HMI tags "Default tag table"
   "DB500_SinaisIhm_ManFrente" : Bool = PLC DB500_SinaisIhm.ManFrente AT %DB500.DBX10.1, 1 s
   "DB500_SinaisIhm_ManDireita" : Bool = PLC DB500_SinaisIhm.ManDireita AT %DB500.DBX10.3, 1 s
   "DB500_SinaisIhm_ManTras" : Bool = PLC DB500_SinaisIhm.ManTras AT %DB500.DBX10.2, 1 s
   "DB500_SinaisIhm_ManEsquerda" : Bool = PLC DB500_SinaisIhm.ManEsquerda AT %DB500.DBX10.4, 1 s
   "DB500_SinaisIhm_ManualAutomatico" : Int = PLC DB500_SinaisIhm.ManualAutomatico AT %DB500.DBW0, 1 s
   "DB500_SinaisIhm_Start" : Bool = PLC DB500_SinaisIhm.Start AT %DB500.DBX2.0, 1 s
   "DB1_DatabaseAgv_Entradas.ScannerWarning" : Bool = PLC DB1_DatabaseAgv.Entradas.ScannerWarning AT %DB1.DBX0.2, 1 s
   "DB1_DatabaseAgv_Entradas.ScannerSafety" : Bool = PLC DB1_DatabaseAgv.Entradas.ScannerSafety AT %DB1.DBX0.3, 1 s
   "DB1_DatabaseAgv_PGV.Module2.PositionY" : DWord = PLC DB1_DatabaseAgv.PGV.Module2.PositionY AT %DB1.DBD10, 1 s
   "DB1_DatabaseAgv_Entradas.BotaoEmergencia" : Bool = PLC DB1_DatabaseAgv.Entradas.BotaoEmergencia AT %DB1.DBX0.1, 1 s
   "DB1_DatabaseAgv_PGV.NaRota" : Bool = PLC DB1_DatabaseAgv.PGV.NaRota AT %DB1.DBX284.0, 1 s
   "DB1_DatabaseAgv_MotorDePasso.OutPuts.ActualPosition" : DInt = PLC DB1_DatabaseAgv.MotorDePasso.OutPuts.ActualPosition AT %DB1.DBD672, 1 s
   "DB3_Memorias_LimiteGiroEsquerda" : Bool = PLC DB3_Memorias.LimiteGiroEsquerda AT %DB3.DBX28.3, 1 s
   "DB3_Memorias_LimiteGiroDireita" : Bool = PLC DB3_Memorias.LimiteGiroDireita AT %DB3.DBX28.2, 1 s
   "DB1_DatabaseAgv_Saidas.Giroflex" : Bool = PLC DB1_DatabaseAgv.Saidas.Giroflex AT %DB1.DBX2.4, 1 s
   "DB1_DatabaseAgv_RFID.Posto" : Int = PLC DB1_DatabaseAgv.RFID.Posto AT %DB1.DBW306, 1 s
   "DB1_DatabaseAgv_PGV.Rota" : Byte = PLC DB1_DatabaseAgv.PGV.Rota AT %DB1.DBB285, 1 s
   "DB500_SinaisIhm_VelocidadeManual" : Int = PLC DB500_SinaisIhm.VelocidadeManual AT %DB500.DBW6, 1 s
   "DB500_SinaisIhm_VelocidadeWarning" : Int = PLC DB500_SinaisIhm.VelocidadeWarning AT %DB500.DBW8, 1 s
   "DB600_AgvSinais_Mensagens_Global" : String[254] = PLC DB600_AgvSinais.Mensagens_Global AT %DB600.DBX836.0, 1 s
   "DB600_AgvSinais_RFID.Tag_Presente" : Bool = PLC DB600_AgvSinais.RFID.Tag_Presente AT %DB600.DBX16.0, 1 s
   "DB600_AgvSinais_RFID.Ready" : Bool = PLC DB600_AgvSinais.RFID.Ready AT %DB600.DBX20.0, 1 s
   "DB600_AgvSinais_RFID.Error" : Bool = PLC DB600_AgvSinais.RFID.Error AT %DB600.DBX16.1, 1 s
   "DB600_AgvSinais_RFID.Code_Error" : Int = PLC DB600_AgvSinais.RFID.Code_Error AT %DB600.DBW18, 1 s
   "DB600_AgvSinais_RFID.Posto" : Int = PLC DB600_AgvSinais.RFID.Posto AT %DB600.DBW8, 1 s
   "DB600_AgvSinais_RFID.Comando" : Int = PLC DB600_AgvSinais.RFID.Comando AT %DB600.DBW10, 1 s
   "DB600_AgvSinais_RFID.Velocidade" : Int = PLC DB600_AgvSinais.RFID.Velocidade AT %DB600.DBW12, 1 s
   "DB600_AgvSinais_RFID.Mensagem" : String[254] = PLC DB600_AgvSinais.RFID.Mensagem AT %DB600.DBX22.0, 1 s
   "DB600_AgvSinais_PGV.PositionData_Y" : Int = PLC DB600_AgvSinais.PGV.PositionData_Y AT %DB600.DBW804, 1 s
   "DB600_AgvSinais_PGV.PositionData_X" : Int = PLC DB600_AgvSinais.PGV.PositionData_X AT %DB600.DBW806, 1 s
   "DB600_AgvSinais_PGV.PositionData_Z" : Int = PLC DB600_AgvSinais.PGV.PositionData_Z AT %DB600.DBW808, 1 s
   "DB600_AgvSinais_PGV.ERR" : Bool = PLC DB600_AgvSinais.PGV.ERR AT %DB600.DBX802.0, 1 s
   "DB600_AgvSinais_PGV.NP" : Bool = PLC DB600_AgvSinais.PGV.NP AT %DB600.DBX802.1, 1 s
   "DB600_AgvSinais_PGV.WRN" : Bool = PLC DB600_AgvSinais.PGV.WRN AT %DB600.DBX802.2, 1 s
   "DB600_AgvSinais_PGV.CA" : Bool = PLC DB600_AgvSinais.PGV.CA AT %DB600.DBX802.3, 1 s
   "DB600_AgvSinais_PGV.FR" : Bool = PLC DB600_AgvSinais.PGV.FR AT %DB600.DBX802.4, 1 s
   "DB600_AgvSinais_PGV.FL" : Bool = PLC DB600_AgvSinais.PGV.FL AT %DB600.DBX802.5, 1 s
   "DB600_AgvSinais_PGV.Mensagem" : String[254] = PLC DB600_AgvSinais.PGV.Mensagem AT %DB600.DBX546.0, 1 s
   "DB600_AgvSinais_Stepping_Motor.Outputs.DriveEnabled" : Bool = PLC DB600_AgvSinais.Stepping_Motor.Outputs.DriveEnabled AT %DB600.DBX284.0, 1 s
   "DB600_AgvSinais_Stepping_Motor.Outputs.Ready" : Bool = PLC DB600_AgvSinais.Stepping_Motor.Outputs.Ready AT %DB600.DBX284.1, 1 s
   "DB600_AgvSinais_Stepping_Motor.Outputs.Warning" : Bool = PLC DB600_AgvSinais.Stepping_Motor.Outputs.Warning AT %DB600.DBX284.2, 1 s
   "DB600_AgvSinais_Stepping_Motor.Outputs.Fault" : Bool = PLC DB600_AgvSinais.Stepping_Motor.Outputs.Fault AT %DB600.DBX284.3, 1 s
   "DB600_AgvSinais_Stepping_Motor.Outputs.SupplyVoltPresent" : Bool = PLC DB600_AgvSinais.Stepping_Motor.Outputs.SupplyVoltPresent AT %DB600.DBX284.4, 1 s
   "DB600_AgvSinais_Stepping_Motor.Outputs.DragError" : Bool = PLC DB600_AgvSinais.Stepping_Motor.Outputs.DragError AT %DB600.DBX284.5, 1 s
   "DB600_AgvSinais_Stepping_Motor.Outputs.HomingValid" : Bool = PLC DB600_AgvSinais.Stepping_Motor.Outputs.HomingValid AT %DB600.DBX284.6, 1 s
   "DB600_AgvSinais_Stepping_Motor.Outputs.StrokeLimitReached" : Bool = PLC DB600_AgvSinais.Stepping_Motor.Outputs.StrokeLimitReached AT %DB600.DBX284.7, 1 s
   "DB600_AgvSinais_Stepping_Motor.Outputs.ActualPosition" : DInt = PLC DB600_AgvSinais.Stepping_Motor.Outputs.ActualPosition AT %DB600.DBD286, 1 s
   "DB600_AgvSinais_Stepping_Motor.Mensagem" : String[254] = PLC DB600_AgvSinais.Stepping_Motor.Mensagem AT %DB600.DBX290.0, 1 s
   "DB600_AgvSinais_Inputs.8DI_24V.I0.1" : Bool = PLC DB600_AgvSinais.Inputs.8DI_24V."I0.1" AT %DB600.DBX0.1, 1 s
   "DB500_SinaisIhm_PostoRfid" : Int = PLC DB500_SinaisIhm.PostoRfid AT %DB500.DBW12, 1 s
   "DB500_SinaisIhm_ComandoRfid" : Int = PLC DB500_SinaisIhm.ComandoRfid AT %DB500.DBW14, 1 s
   "DB500_SinaisIhm_VelocidadeRfid" : Int = PLC DB500_SinaisIhm.VelocidadeRfid AT %DB500.DBW16, 1 s
   "DB500_SinaisIhm_ProcessoRfid" : Int = PLC DB500_SinaisIhm.ProcessoRfid AT %DB500.DBW18, 1 s
   "DB1_DatabaseAgv_RFID.Inputs.Start" : Bool = PLC DB1_DatabaseAgv.RFID.Inputs.Start AT %DB1.DBX286.1, 1 s
   "DB1_DatabaseAgv_RFID.Inputs.Command" : Int = PLC DB1_DatabaseAgv.RFID.Inputs.Command AT %DB1.DBW290, 1 s
   "DB1_DatabaseAgv_RFID.Comando" : Int = PLC DB1_DatabaseAgv.RFID.Comando AT %DB1.DBW308, 1 s
   "DB1_DatabaseAgv_RFID.Velocidade" : Int = PLC DB1_DatabaseAgv.RFID.Velocidade AT %DB1.DBW310, 1 s
   "DB1_DatabaseAgv_RFID.Processo" : Int = PLC DB1_DatabaseAgv.RFID.Processo AT %DB1.DBW312, 1 s
   "DB600_AgvSinais_Inputs.8DI_24V.I0.0" : Bool = PLC DB600_AgvSinais.Inputs.8DI_24V."I0.0" AT %DB600.DBX0.0, 1 s
   "DB600_AgvSinais_Inputs.8DI_24V.I0.2" : Bool = PLC DB600_AgvSinais.Inputs.8DI_24V."I0.2" AT %DB600.DBX0.2, 1 s
   "DB600_AgvSinais_Inputs.8DI_24V.I0.3" : Bool = PLC DB600_AgvSinais.Inputs.8DI_24V."I0.3" AT %DB600.DBX0.3, 1 s
   "DB600_AgvSinais_Inputs.8DI_24V.I0.4" : Bool = PLC DB600_AgvSinais.Inputs.8DI_24V."I0.4" AT %DB600.DBX0.4, 1 s
   "DB600_AgvSinais_Inputs.8DI_24V.I0.5" : Bool = PLC DB600_AgvSinais.Inputs.8DI_24V."I0.5" AT %DB600.DBX0.5, 1 s
   "DB600_AgvSinais_Inputs.8DI_24V.I0.6" : Bool = PLC DB600_AgvSinais.Inputs.8DI_24V."I0.6" AT %DB600.DBX0.6, 1 s
   "DB600_AgvSinais_Inputs.8DI_24V.I0.7" : Bool = PLC DB600_AgvSinais.Inputs.8DI_24V."I0.7" AT %DB600.DBX0.7, 1 s
   "DB600_AgvSinais_Outputs.8DO_24V.Q0.0" : Bool = PLC DB600_AgvSinais.Outputs.8DO_24V."Q0.0" AT %DB600.DBX2.0, 1 s
   "DB600_AgvSinais_Outputs.8DO_24V.Q0.1" : Bool = PLC DB600_AgvSinais.Outputs.8DO_24V."Q0.1" AT %DB600.DBX2.1, 1 s
   "DB600_AgvSinais_Outputs.8DO_24V.Q0.2" : Bool = PLC DB600_AgvSinais.Outputs.8DO_24V."Q0.2" AT %DB600.DBX2.2, 1 s
   "DB600_AgvSinais_Outputs.8DO_24V.Q0.3" : Bool = PLC DB600_AgvSinais.Outputs.8DO_24V."Q0.3" AT %DB600.DBX2.3, 1 s
   "DB600_AgvSinais_Outputs.8DO_24V.Q0.4" : Bool = PLC DB600_AgvSinais.Outputs.8DO_24V."Q0.4" AT %DB600.DBX2.4, 1 s
   "DB600_AgvSinais_Outputs.8DO_24V.Q0.5" : Bool = PLC DB600_AgvSinais.Outputs.8DO_24V."Q0.5" AT %DB600.DBX2.5, 1 s
   "DB600_AgvSinais_Outputs.8DO_24V.Q0.6" : Bool = PLC DB600_AgvSinais.Outputs.8DO_24V."Q0.6" AT %DB600.DBX2.6, 1 s
   "DB600_AgvSinais_Outputs.8DO_24V.Q0.7" : Bool = PLC DB600_AgvSinais.Outputs.8DO_24V."Q0.7" AT %DB600.DBX2.7, 1 s
   "DB600_AgvSinais_Outputs.2AO x U ST.QW750" : Word = PLC DB600_AgvSinais.Outputs."2AO x U ST".QW750 AT %DB600.DBW4, 1 s
   "DB600_AgvSinais_Outputs.2AO x U ST.QW752" : Word = PLC DB600_AgvSinais.Outputs."2AO x U ST".QW752 AT %DB600.DBW6, 1 s
   "DB600_AgvSinais_Stepping_Motor.Inputs.Enabla_Drive" : Bool = PLC DB600_AgvSinais.Stepping_Motor.Inputs.Enabla_Drive AT %DB600.DBX278.0, 1 s
   "DB600_AgvSinais_Stepping_Motor.Inputs.Stop" : Bool = PLC DB600_AgvSinais.Stepping_Motor.Inputs.Stop AT %DB600.DBX278.1, 1 s
   "DB600_AgvSinais_Stepping_Motor.Inputs.Start Task" : Bool = PLC DB600_AgvSinais.Stepping_Motor.Inputs."Start Task" AT %DB600.DBX278.2, 1 s
   "DB600_AgvSinais_Stepping_Motor.Inputs.Opm" : Int = PLC DB600_AgvSinais.Stepping_Motor.Inputs.Opm AT %DB600.DBW280, 1 s
   "DB1_DatabaseAgv_RFID.Inputs.Reset" : Bool = PLC DB1_DatabaseAgv.RFID.Inputs.Reset AT %DB1.DBX286.2, 1 s
   "DB1_DatabaseAgv_MotorDePasso.Inputs.ResetFault" : Bool = PLC DB1_DatabaseAgv.MotorDePasso.Inputs.ResetFault AT %DB1.DBX622.4, 1 s
   "DB1_DatabaseAgv_MotorDePasso.Inputs.StartHoming" : Bool = PLC DB1_DatabaseAgv.MotorDePasso.Inputs.StartHoming AT %DB1.DBX626.1, 1 s
   "DB600_AgvSinais_Alarms[0]" : Int = PLC DB600_AgvSinais.Alarms[0] AT %DB600.DBW1092, 1 s
   "DB600_AgvSinais_DateHora" : Date_And_Time = PLC DB600_AgvSinais.DateHora AT %DB600.DBX828.0, 1 s
   "DB703_ControleTakt_Out_Get_Error" : Bool = PLC DB703_ControleTakt.Out_Get_Error AT %DB703.DBX30.0, 1 s
   "DB703_ControleTakt_Out_Set_Erro" : Bool = PLC DB703_ControleTakt.Out_Set_Erro AT %DB703.DBX34.0, 1 s
   "DB703_ControleTakt_Out_Get_Status" : Word = PLC DB703_ControleTakt.Out_Get_Status AT %DB703.DBW32, 1 s
   "DB703_ControleTakt_Out_Set_Status" : Word = PLC DB703_ControleTakt.Out_Set_Status AT %DB703.DBW36, 1 s
   "DB500_SinaisIhm_VelocidadeAtual" : Int = PLC DB500_SinaisIhm.VelocidadeAtual AT %DB500.DBW24, 1 s
   "DB500_SinaisIhm_VelocidadeAutomatico" : Int = PLC DB500_SinaisIhm.VelocidadeAutomatico AT %DB500.DBW22, 1 s
   "DB500_SinaisIhm_ConexaoTakt" : Bool = PLC DB500_SinaisIhm.ConexaoTakt AT %DB500.DBX10.5, 1 s
   "DB500_SinaisIhm_ConectarTakt" : Int = PLC DB500_SinaisIhm.ConectarTakt AT %DB500.DBW26, 1 s
   "DB3_Memorias_StartStop" : Bool = PLC DB3_Memorias.StartStop AT %DB3.DBX0.0, 1 s
   "DB500_SinaisIhm_ResetFalha_Rfid" : Bool = PLC DB500_SinaisIhm.ResetFalha_Rfid AT %DB500.DBX28.0, 1 s
   "DB420_LeituraRfid_RfidLeitura[3]" : Int = PLC DB420_LeituraRfid.RfidLeitura[3] AT %DB420.DBW6, 1 s

discrete alarms
   1: 'AGV FORA DA ROTA', class Warnings, trigger "DB600_AgvSinais_Alarms[0]" bit 1
   2: 'AREA DE ATENÇÃO DO SCANNER INFRINGIDA', class Warnings, trigger "DB600_AgvSinais_Alarms[0]" bit 2
   3: 'AREA DE SEGURANÇA DO SCANNER INFRINGIDA', class Warnings, trigger "DB600_AgvSinais_Alarms[0]" bit 3
   4: 'EMERGENCIA PRECIONADO', class Warnings, trigger "DB600_AgvSinais_Alarms[0]" bit 4
   5: 'FALHA NO MOTOR DE PASSO', class Warnings, trigger "DB600_AgvSinais_Alarms[0]" bit 5
   6: 'CHAVE DO MOTOR DE TRAÇÃO DESLIGADA', class Warnings, trigger "DB600_AgvSinais_Alarms[0]" bit 6
   7: 'RFID FORA DA REDE', class Warnings, trigger "DB600_AgvSinais_Alarms[0]" bit 7
   9: 'PGV FORA DA REDE', class Warnings, trigger "DB600_AgvSinais_Alarms[0]" bit 8
   10: 'MOTOR DE PASSO FORA DA REDE', class Warnings, trigger "DB600_AgvSinais_Alarms[0]" bit 9
   11: 'SEM COMUNICAÇÃO COM O TAKT', class Warnings, trigger "DB600_AgvSinais_Alarms[0]" bit 10
   12: 'EMERGENCIA ACIONADO NA LINHA DE SKD', class Warnings, trigger "DB600_AgvSinais_Alarms[0]" bit 12

screen "00_Home" 320x240, template "Template_1"
   Softkey "Softkey_F2" at 0,0 size 0x0
      on KeyDown: ActivateScreen("01_Manual", 0); SetTag("DB500_SinaisIhm_ManualAutomatico", 1); ResetBit("DB500_SinaisIhm_Start")
   Softkey "Softkey_F5" at 0,0 size 0x0
      on KeyDown: SetTag("DB500_SinaisIhm_ManualAutomatico", 2)
   Softkey "Softkey_F6" at 0,0 size 0x0
      on KeyDown: SetBit("DB500_SinaisIhm_Start")
   GraphicView "Graphic view_2" at 109,59 size 115x100; Picture "Graphic_15"
      Visibility <- "DB1_DatabaseAgv_Entradas.BotaoEmergencia"
   Rectangle "Rectangle_2" at 82,66 size 43x87
      Visibility <- "DB1_DatabaseAgv_Entradas.BotaoEmergencia"
      Appearance <- "DB1_DatabaseAgv_Entradas.ScannerSafety"
   Circle "Circle_3" at 148,102 size 17x17
      Visibility <- "DB1_DatabaseAgv_Entradas.BotaoEmergencia"
      Appearance <- "DB1_DatabaseAgv_Saidas.Giroflex"
   GraphicView "Graphic view_1" at 125,78 size 146x65; Picture "Graphic_14"
      Visibility <- "DB1_DatabaseAgv_Entradas.BotaoEmergencia"
   Circle "Circle_4" at 149,103 size 17x17
      Visibility <- "DB1_DatabaseAgv_Entradas.BotaoEmergencia"
      Appearance <- "DB1_DatabaseAgv_Saidas.Giroflex"
   Button "Button_1" at 54,202 size 52x38; TextOff 'MANUAL'
      on Press: ActivateScreen("01_Manual", 0); SetTag("DB500_SinaisIhm_ManualAutomatico", 1); ResetBit("DB500_SinaisIhm_Start")
   Button "Button_2" at 213,202 size 52x38; TextOff 'AUTOMA TICO'
      on Press: SetTag("DB500_SinaisIhm_ManualAutomatico", 2)
      Appearance <- "DB500_SinaisIhm_ManualAutomatico"
   Button "Button_3" at 266,202 size 52x38; TextOff 'START'
      on Press: SetBit("DB500_SinaisIhm_Start")
      Appearance <- "DB3_Memorias_StartStop"
   IOField "I/O field_1" at 5,28 size 35x20; FormatPattern 99
      ProcessValue <- "DB1_DatabaseAgv_RFID.Posto"
   TextField "Text field_9" at 41,30 size 38x13; Text 'POSTO'
   Circle "Circle_5" at 5,72 size 13x13
      Appearance <- "DB1_DatabaseAgv_Entradas.ScannerWarning"
   Circle "Circle_6" at 5,91 size 13x13
      Appearance <- "DB1_DatabaseAgv_Entradas.ScannerSafety"
   TextField "Text field_8" at 21,72 size 52x13; Text 'WARNING'
   TextField "Text field_13" at 25,91 size 42x13; Text 'SAFETY'
   Circle "Circle_1" at 83,32 size 13x13
      Appearance <- "DB1_DatabaseAgv_PGV.Module2.PositionY"
   TextField "Text field_4" at 103,25 size 42x24; Text 'AGV NA ROTA'
   Circle "Circle_2" at 231,33 size 23x23
      Appearance <- "DB500_SinaisIhm_ConectarTakt"
   IOField "I/O field_4" at 130,1 size 186x15; FormatPattern 9999999999999999999999999999999999999999
      ProcessValue <- "DB600_AgvSinais_DateHora"
   TextField "Text field_10" at 265,26 size 53x35; Text 'CONEXÃO COM O TAKT'
   IOField "I/O field_5" at 0,175 size 319x27; FormatPattern ????????????????????????????????????????????????????????????????????????????????
      ProcessValue <- "DB600_AgvSinais_Mensagens_Global"
   Button "Button_4" at 160,202 size 52x38; TextOff 'PARA METROS'
      on Press: ActivateScreen("02_Parametros", 0)
   Button "Button_5" at 107,202 size 52x38; TextOff 'MANU TENÇÂO'
      on Press: ActivateScreen("03_Manutecao", 0)
   IOField "I/O field_2" at 236,153 size 63x17; FormatPattern 99; Unit  M/MIN
      ProcessValue <- "DB500_SinaisIhm_VelocidadeAtual"
   Softkey "Softkey_F4" at 0,0 size 0x0
      on KeyDown: ActivateScreen("02_Parametros", 0)
   Softkey "Softkey_F3" at 0,0 size 0x0
      on KeyUp: ActivateScreen("03_Manutecao", 0)

Template "Template_1" 320x240
   Softkey "Softkey_F1" at 0,0 size 0x0; SoftkeyImage "Home"
      on KeyDown: ActivateScreen("00_Home", 0)
   TextField "Template_Text field_1" at 4,0 size 60x15; Text 'AGV75790'

screen "01_Manual" 320x240, template "Template_1"
   Button "Button_1" at 9,96 size 75x26; TextOff 'FRENTE'
      on Press: SetBit("DB500_SinaisIhm_ManFrente")
      on Release: ResetBit("DB500_SinaisIhm_ManFrente")
   Button "Button_2" at 244,97 size 75x26; TextOff 'TRÁS'
      on Release: ResetBit("DB500_SinaisIhm_ManTras")
      on Press: SetBit("DB500_SinaisIhm_ManTras")
   Button "Button_3" at 128,28 size 75x26; TextOff 'DIREITA'
      on Release: ResetBit("DB500_SinaisIhm_ManDireita")
      on Press: SetBit("DB500_SinaisIhm_ManDireita")
   Button "Button_4" at 130,159 size 75x26; TextOff 'ESQUERDA'
      on Release: ResetBit("DB500_SinaisIhm_ManEsquerda")
      on Press: SetBit("DB500_SinaisIhm_ManEsquerda")
   GraphicView "Graphic view_2" at 112,58 size 115x100; Picture "Graphic_15"
      Visibility <- "DB1_DatabaseAgv_Entradas.BotaoEmergencia"
   Rectangle "Rectangle_1" at 129,76 size 102x63
      Visibility <- "DB1_DatabaseAgv_Entradas.BotaoEmergencia"
   Line "Line_1" at 129,106 size 102x0
      Visibility <- "DB1_DatabaseAgv_Entradas.BotaoEmergencia"
   Rectangle "Rectangle_2" at 197,114 size 28x19
      Visibility <- "DB1_DatabaseAgv_Entradas.BotaoEmergencia"
   Circle "Circle_1" at 140,116 size 12x12
      Visibility <- "DB1_DatabaseAgv_Entradas.BotaoEmergencia"
   Circle "Circle_2" at 161,116 size 12x12
      Visibility <- "DB1_DatabaseAgv_Entradas.BotaoEmergencia"
      Appearance <- "DB1_DatabaseAgv_Entradas.BotaoEmergencia"
   Rectangle "Rectangle_3" at 111,76 size 19x63
      Visibility <- "DB1_DatabaseAgv_Entradas.BotaoEmergencia"
   Circle "Circle_3" at 111,99 size 17x17
      Visibility <- "DB1_DatabaseAgv_Entradas.BotaoEmergencia"
      Appearance <- "DB1_DatabaseAgv_Saidas.Giroflex"
   Rectangle "Rectangle_4" at 101,98 size 10x19
      Visibility <- "DB1_DatabaseAgv_Entradas.BotaoEmergencia"
   Circle "Circle_4" at 89,98 size 19x19
      Visibility <- "DB1_DatabaseAgv_Entradas.BotaoEmergencia"
   TextField "Text field_3" at 25,11 size 50x14; Text 'SCANNER'
   TextField "Text field_4" at 100,11 size 164x15; Text 'LIMITE DE GIRO ALCANÇADO'
      Visibility <- "DB3_Memorias_LimiteGiroDireita"
   TextField "Text field_5" at 91,186 size 165x15; Text 'LIMITE DE GIRO ALCANÇADO'
      Visibility <- "DB3_Memorias_LimiteGiroEsquerda"
   IOField "I/O field_5" at 56,202 size 263x37; FormatPattern ????????????????????????????????????????????????????????????????????????????????
      ProcessValue <- "DB600_AgvSinais_Mensagens_Global"
   TextField "Text field_6" at 36,65 size 42x24; Text 'AGV NA ROTA'
   Circle "Circle_5" at 16,30 size 13x13
      Appearance <- "DB1_DatabaseAgv_Entradas.ScannerWarning"
   Circle "Circle_6" at 16,49 size 13x13
      Appearance <- "DB1_DatabaseAgv_Entradas.ScannerSafety"
   TextField "Text field_8" at 32,30 size 52x13; Text 'WARNING'
   TextField "Text field_13" at 36,49 size 42x13; Text 'SAFETY'
   Circle "Circle_7" at 16,69 size 13x13
      Appearance <- "DB1_DatabaseAgv_PGV.Module2.PositionY"
   TextField "Text field_11" at 19,139 size 55x24; Text 'ACTUAL POSITION'
   IOField "I/O field_2" at 6,167 size 73x30; FormatPattern s9999999999
      ProcessValue <- "DB1_DatabaseAgv_MotorDePasso.OutPuts.ActualPosition"

screen "02_Parametros" 320x240, template "Template_1"
   TextField "Text field_9" at 72,4 size 172x20; Text 'TELA DE PARAMETROS'
   TextField "Text field_1" at 5,27 size 61x24; Text 'MODO DE OPERAÇÃO'
   Switch "Switch_1" at 2,55 size 64x32; TextOn 'MODO TAKT'; CaptionText 'Switch'; TextOff 'MODO MANUAL'
      on SwitchOn: SetBit("DB500_SinaisIhm_ConexaoTakt")
      on SwitchOff: ResetBit("DB500_SinaisIhm_ConexaoTakt")
      Appearance <- "DB500_SinaisIhm_ConexaoTakt"
   Switch "Switch_2" at 109,52 size 64x36; TextOn 'LINHA SKD'; CaptionText 'Switch'; TextOff 'LINHA ECU'
      on SwitchOff: SetTag("DB1_DatabaseAgv_PGV.Rota", 10)
      on SwitchOn: SetTag("DB1_DatabaseAgv_PGV.Rota", 1)
      ProcessValue <- "DB1_DatabaseAgv_PGV.Rota"
      Appearance <- "DB1_DatabaseAgv_PGV.Rota"
   TextField "Text field_16" at 118,39 size 22x13; Text 'ECU'
   TextField "Text field_17" at 143,39 size 22x13; Text 'SKD'
   TextField "Text field_18" at 138,39 size 10x13; Text '/'
   TextField "Text field_2" at 89,26 size 114x13; Text 'LINHA DE TRABALHO'
   Circle "Circle_1" at 203,50 size 23x23
      Appearance <- "DB500_SinaisIhm_ConectarTakt"
   TextField "Text field_3" at 236,42 size 53x35; Text 'CONEXÃO COM O TAKT'
   Switch "Toggle_Horizontal_GN" at 104,97 size 87x58; CaptionText 'Switch'; TextOff '0'; TextOn '1'; PictureOff "Toggle_Horizontal_GN_Off_256c"; PictureOn "Toggle_Horizontal_GN_On_256c"
      on SwitchOff: SetTag("DB1_DatabaseAgv_PGV.Rota", 10)
      on SwitchOn: SetTag("DB1_DatabaseAgv_PGV.Rota", 1)
      ProcessValue <- "DB1_DatabaseAgv_PGV.Rota"
   Button "Button_7" at 3,124 size 63x29; TextOff 'PLC'
      on Release: ActivateScreen("12_Alarms", 0)
   TextField "Text field_4" at 4,96 size 84x24; Text 'ACESSO A TELA DE DIAGNOSE'
   TextField "Text field_5" at 215,87 size 75x13; Text 'VELOCIDADES'
   TextField "Text field_6" at 222,102 size 59x13; Text 'WARNNING'
   TextField "Text field_7" at 228,135 size 47x13; Text 'MANUAL'
   IOField "I/O field_1" at 232,115 size 35x20; FormatPattern 99
      ProcessValue <- "DB500_SinaisIhm_VelocidadeWarning"
   IOField "I/O field_2" at 232,151 size 35x20; FormatPattern 99
      ProcessValue <- "DB500_SinaisIhm_VelocidadeManual"
   TextField "Text field_8" at 214,171 size 76x13; Text 'AUTOMATICO'
   IOField "I/O field_3" at 232,187 size 35x20; FormatPattern 99
      ProcessValue <- "DB420_LeituraRfid_RfidLeitura[3]"

screen "03_Manutecao" 320x240, template "Template_1"
   TextField "Text field_9" at 75,3 size 175x20; Text 'TELA DE MANUTENÇÃO'
   Button "Button_1" at 137,55 size 82x29; TextOff 'RFID'
      on Release: ActivateScreen("04_RfidStatus", 0)
   Button "Button_4" at 227,55 size 82x29; TextOff 'PGV'
      on Release: ActivateScreen("05_PgvStatus", 0)
   Button "Button_5" at 227,93 size 82x29; TextOff 'IO-LINK'
      on Release: ActivateScreen("07_IoLinkStatus", 0)
   Button "Button_6" at 137,93 size 82x29; TextOff 'MOTOR PASSO'
      on Release: ActivateScreen("06_Status_Saida_MotorDePasso", 0)
   Button "Button_7" at 227,129 size 82x29; TextOff 'PLC'
      on Release: ActivateScreen("08_PlcStatus", 0)
   TextField "Text field_1" at 183,27 size 91x15; Text 'STATUS DO AGV'
   TextField "Text field_2" at 24,27 size 57x15; Text 'AUXILIAR'
   Button "Button_2" at 15,54 size 82x29; TextOff 'CONFIG. TAGS RFID'
      on Release: ActivateScreen("09_ConfigTagsRfid", 0)
   Button "Button_3" at 15,90 size 82x29; TextOff 'DIFFERENT JOBS'
   IOField "I/O field_5" at 58,202 size 261x36; FormatPattern ????????????????????????????????????????????
      ProcessValue <- "DB600_AgvSinais_Mensagens_Global"
   Button "Button_8" at 137,129 size 82x29; TextOff 'TAKT'
      on Release: ActivateScreen("14_StatusTakt", 0)

screen "04_RfidStatus" 320x240, template "Template_2"
   TextField "Text field_5" at 72,3 size 164x18; Text 'TELA DE STATUS DO RFID'
   GraphicView "Graphic view_1" at 8,33 size 113x90; Picture "Graphic_11"
   Circle "Circle_1" at 197,39 size 16x16
      Appearance <- "DB600_AgvSinais_RFID.Tag_Presente"
   TextField "Text field_2" at 217,40 size 79x13; Text 'TAG PRESENTE'
   Circle "Circle_2" at 197,61 size 16x16
      Appearance <- "DB600_AgvSinais_RFID.Ready"
   TextField "Text field_3" at 217,62 size 37x13; Text 'READY'
   Circle "Circle_3" at 197,83 size 16x16
      Appearance <- "DB600_AgvSinais_RFID.Error"
   TextField "Text field_4" at 217,84 size 37x13; Text 'ERROR'
   TextField "Text field_6" at 210,106 size 62x24; Text 'CODIGO DO ERROR'
   IOField "I/O field_1" at 212,133 size 54x24; FormatPattern 9999
      ProcessValue <- "DB600_AgvSinais_RFID.Code_Error"
   Circle "Circle_4" at 16,68 size 16x16
      Appearance <- "DB600_AgvSinais_RFID.Tag_Presente"
   Circle "Circle_5" at 56,88 size 16x16
      Appearance <- "DB600_AgvSinais_RFID.Ready"
   IOField "I/O field_2" at 0,127 size 35x20; FormatPattern 99
      ProcessValue <- "DB600_AgvSinais_RFID.Posto"
   IOField "I/O field_3" at 0,152 size 35x20; FormatPattern 99
      ProcessValue <- "DB600_AgvSinais_RFID.Comando"
   TextField "Text field_9" at 40,132 size 38x13; Text 'POSTO'
   TextField "Text field_10" at 40,157 size 56x13; Text 'COMANDO'
   IOField "I/O field_4" at 0,177 size 35x20; FormatPattern 99
      ProcessValue <- "DB600_AgvSinais_RFID.Velocidade"
   TextField "Text field_14" at 40,182 size 69x13; Text 'VELOCIDADE'
   IOField "I/O field_5" at 109,202 size 210x35; FormatPattern ????????????????????????????????????????????
      ProcessValue <- "DB600_AgvSinais_RFID.Mensagem"
   Button "Button_1" at 120,167 size 71x32; TextOff 'RESET FALHA'
      on Press: SetBit("DB500_SinaisIhm_ResetFalha_Rfid")
      on Release: ResetBit("DB500_SinaisIhm_ResetFalha_Rfid")

screen "05_PgvStatus" 320x240, template "Template_2"
   TextField "Text field_5" at 77,5 size 156x18; Text 'TELA DE STATUS DO PGV'
   GraphicView "Graphic view_1" at 5,69 size 72x85; Picture "Graphic_12"
   Circle "Circle_4" at 189,38 size 16x16
      Appearance <- "DB600_AgvSinais_PGV.ERR"
   TextField "Text field_6" at 209,39 size 30x13; Text 'ERRO'
   TextField "Text field_2" at 5,32 size 61x13; Text 'POSIÇÃO X'
   TextField "Text field_3" at 93,82 size 61x13; Text 'POSIÇÃO Y'
   TextField "Text field_4" at 5,158 size 60x13; Text 'POSIÇÃO Z'
   IOField "I/O field_1" at 6,48 size 67x23; FormatPattern 99999
      ProcessValue <- "DB600_AgvSinais_PGV.PositionData_X"
   IOField "I/O field_2" at 93,104 size 67x23; FormatPattern 99999
      ProcessValue <- "DB600_AgvSinais_PGV.PositionData_Y"
   IOField "I/O field_3" at 0,173 size 67x23; FormatPattern 99999
      ProcessValue <- "DB600_AgvSinais_PGV.PositionData_Z"
   Circle "Circle_1" at 189,59 size 16x16
      Appearance <- "DB600_AgvSinais_PGV.NP"
   TextField "Text field_8" at 209,60 size 50x13; Text 'NA ROTA'
   Circle "Circle_2" at 189,80 size 16x16
      Appearance <- "DB600_AgvSinais_PGV.WRN"
   TextField "Text field_9" at 209,81 size 52x13; Text 'WARNING'
   Circle "Circle_3" at 189,101 size 16x16
      Appearance <- "DB600_AgvSinais_PGV.CA"
   TextField "Text field_10" at 209,102 size 82x12; Text 'QR CODE PRESENTE'
   Circle "Circle_5" at 189,122 size 16x16
      Appearance <- "DB600_AgvSinais_PGV.FR"
   TextField "Text field_11" at 209,123 size 87x13; Text 'SIGA A DIREITA'
   Circle "Circle_6" at 189,143 size 16x16
      Appearance <- "DB600_AgvSinais_PGV.FL"
   TextField "Text field_12" at 209,144 size 87x13; Text 'SIGA A DIREITA'
   IOField "I/O field_5" at 109,202 size 210x35; FormatPattern ????????????????????????????????????????????
      ProcessValue <- "DB600_AgvSinais_PGV.Mensagem"

screen "06_Status_Saida_MotorDePasso" 320x240, template "Template_2"
   TextField "Text field_5" at 79,2 size 188x18; Text 'STATUS DO MOTOR DE PASSO'
   GraphicView "Graphic view_1" at 4,61 size 95x85; Picture "Graphic_13"
   Circle "Circle_1" at 108,32 size 16x16
      Appearance <- "DB600_AgvSinais_Stepping_Motor.Outputs.DriveEnabled"
   TextField "Text field_2" at 128,33 size 52x13; Text 'DRIVE ON'
   Circle "Circle_2" at 108,52 size 16x16
      Appearance <- "DB600_AgvSinais_Stepping_Motor.Outputs.Ready"
   TextField "Text field_3" at 128,53 size 37x13; Text 'READY'
   Circle "Circle_3" at 108,72 size 16x16
      Appearance <- "DB600_AgvSinais_Stepping_Motor.Outputs.Warning"
   TextField "Text field_4" at 128,73 size 52x13; Text 'WARNING'
   Circle "Circle_4" at 108,92 size 16x16
      Appearance <- "DB600_AgvSinais_Stepping_Motor.Outputs.Fault"
   TextField "Text field_6" at 128,93 size 36x13; Text 'FAULT'
   Circle "Circle_5" at 108,112 size 16x16
      Appearance <- "DB600_AgvSinais_Stepping_Motor.Outputs.SupplyVoltPresent"
   TextField "Text field_8" at 128,113 size 99x13; Text 'TENSÃO PRESENTE'
   Circle "Circle_6" at 108,132 size 16x16
      Appearance <- "DB600_AgvSinais_Stepping_Motor.Outputs.DragError"
   TextField "Text field_9" at 128,133 size 69x13; Text 'DRAG ERROR'
   Circle "Circle_7" at 108,152 size 16x16
      Appearance <- "DB600_AgvSinais_Stepping_Motor.Outputs.HomingValid"
   TextField "Text field_10" at 128,153 size 64x13; Text 'HOMING OK'
   TextField "Text field_11" at 247,30 size 55x24; Text 'ACTUAL POSITION'
   IOField "I/O field_1" at 234,58 size 73x30; FormatPattern s9999999999
      ProcessValue <- "DB600_AgvSinais_Stepping_Motor.Outputs.ActualPosition"
   Circle "Circle_8" at 108,170 size 16x16
      Appearance <- "DB600_AgvSinais_Stepping_Motor.Outputs.StrokeLimitReached"
   TextField "Text field_12" at 128,171 size 84x13; Text 'STROKE LIMITE'
   Button "Button_1" at 233,124 size 76x32; TextOff 'PROXIMA PAGINA'
      on Release: ActivateScreen("11_InStatusMotorDePasso", 0)
   IOField "I/O field_5" at 110,201 size 206x35; FormatPattern ????????????????????????????????????????????
      ProcessValue <- "DB600_AgvSinais_Stepping_Motor.Mensagem"

screen "07_IoLinkStatus" 320x240, template "Template_2"
   GraphicView "Graphic view_1" at 138,31 size 58x158; Picture "Graphic_5"
   TextField "Text field_5" at 76,3 size 207x15; Text 'TELA DE STATUS DO MASTER IO-LINK'
   IOField "I/O field_5" at 109,202 size 209x36; FormatPattern ????????????????????????????????????????????
      ProcessValue <- "DB600_AgvSinais_Mensagens_Global"
   Circle "Circle_3" at 12,65 size 17x17
      Appearance <- "DB600_AgvSinais_Inputs.8DI_24V.I0.1"
   TextField "Text field_3" at 33,67 size 30x13; Text 'I/O 2'
   Circle "Circle_4" at 12,83 size 17x17
      Appearance <- "DB600_AgvSinais_Inputs.8DI_24V.I0.1"
   TextField "Text field_4" at 33,85 size 30x13; Text 'I/O 4'
   Circle "Circle_5" at 12,106 size 17x17
      Appearance <- "DB600_AgvSinais_Inputs.8DI_24V.I0.1"
   TextField "Text field_6" at 33,108 size 30x13; Text 'I/O 2'
   Circle "Circle_6" at 12,124 size 17x17
      Appearance <- "DB600_AgvSinais_Inputs.8DI_24V.I0.1"
   TextField "Text field_7" at 33,126 size 30x13; Text 'I/O 4'
   Circle "Circle_7" at 12,147 size 17x17
      Appearance <- "DB600_AgvSinais_Inputs.8DI_24V.I0.1"
   TextField "Text field_8" at 33,149 size 30x13; Text 'I/O 2'
   Circle "Circle_8" at 12,165 size 17x17
      Appearance <- "DB600_AgvSinais_Inputs.8DI_24V.I0.1"
   TextField "Text field_9" at 33,167 size 30x13; Text 'I/O 4'
   Circle "Circle_11" at 244,70 size 17x17
      Appearance <- "DB600_AgvSinais_Inputs.8DI_24V.I0.1"
   TextField "Text field_12" at 265,72 size 30x13; Text 'I/O 2'
   Circle "Circle_12" at 244,88 size 17x17
      Appearance <- "DB600_AgvSinais_Inputs.8DI_24V.I0.1"
   TextField "Text field_13" at 265,90 size 30x13; Text 'I/O 4'
   Circle "Circle_13" at 244,111 size 17x17
      Appearance <- "DB600_AgvSinais_Inputs.8DI_24V.I0.1"
   TextField "Text field_14" at 265,113 size 30x13; Text 'I/O 2'
   Circle "Circle_14" at 244,129 size 17x17
      Appearance <- "DB600_AgvSinais_Inputs.8DI_24V.I0.1"
   TextField "Text field_15" at 265,131 size 30x13; Text 'I/O 4'
   Circle "Circle_15" at 244,152 size 17x17
      Appearance <- "DB600_AgvSinais_Inputs.8DI_24V.I0.1"
   TextField "Text field_16" at 265,154 size 30x13; Text 'I/O 2'
   Circle "Circle_16" at 244,170 size 17x17
      Appearance <- "DB600_AgvSinais_Inputs.8DI_24V.I0.1"
   TextField "Text field_17" at 265,172 size 30x13; Text 'I/O 4'
   Button "Button_1" at 8,26 size 65x29; TextOff 'RFID'
      on Release: ActivateScreen("04_RfidStatus", 0)
   Button "Button_6" at 243,32 size 64x29; TextOff 'MOTOR PASSO'
      on Release: ActivateScreen("06_Status_Saida_MotorDePasso", 0)
   Button "Button_4" at 135,27 size 66x165; TextOff 'Text'
      on Release: ActivateScreen("10_InOutStatus", 0)
   Softkey "Softkey_F6" at 0,0 size 0x0
      on KeyDown: function_ee5b8808("Button_4")
      on KeyUp: function_f101fd67("Button_4")

screen "08_PlcStatus" 320x240, template "Template_2"
   GraphicView "Graphic view_1" at 10,40 size 291x147; Picture "Graphic_4"
   Button "Button_2" at 226,41 size 24x146; TextOff 'Text'
      on Release: ActivateScreen("10_InOutStatus", 0)
   Button "Button_3" at 251,41 size 24x146; TextOff 'Text'
      on Release: ActivateScreen("10_InOutStatus", 0)
   Button "Button_4" at 276,41 size 25x146; TextOff 'Text'
      on Release: ActivateScreen("10_InOutStatus", 0)
   Button "Button_7" at 111,201 size 82x29; TextOff 'ALARMES'
      on Release: ActivateScreen("12_Alarms", 0)
   Button "Button_1" at 226,201 size 82x29; TextOff 'DIAGNOSE'
      on Release: ActivateScreen("13_Diagnose", 0)
   TextField "Text field_5" at 72,6 size 154x18; Text 'TELA DE STATUS DO PLC'
   Softkey "Softkey_F4" at 0,0 size 0x0
      on KeyDown: function_ee5b8808("Button_2")
      on KeyUp: function_f101fd67("Button_2")
   Softkey "Softkey_F5" at 0,0 size 0x0
      on KeyDown: function_ee5b8808("Button_3")
      on KeyUp: function_f101fd67("Button_3")
   Softkey "Softkey_F6" at 0,0 size 0x0
      on KeyDown: function_ee5b8808("Button_4")
      on KeyUp: function_f101fd67("Button_4")

screen "09_ConfigTagsRfid" 320x240, template "Template_2"
   IOField "I/O field_2" at 124,114 size 35x20; FormatPattern 999
      ProcessValue <- "DB500_SinaisIhm_ComandoRfid"
   TextField "Text field_9" at 63,116 size 52x13; Text 'ESTAÇÃO'
   TextField "Text field_10" at 164,119 size 56x13; Text 'COMANDO'
   IOField "I/O field_3" at 228,117 size 35x20; FormatPattern 999
      ProcessValue <- "DB500_SinaisIhm_VelocidadeRfid"
   TextField "Text field_14" at 266,120 size 51x13; Text 'VELOCID.'
   Switch "Switch_1" at 17,168 size 78x32; TextOn 'ESCRITA'; CaptionText 'Switch'; TextOff 'LEITURA'
      on SwitchOff: SetTag("DB1_DatabaseAgv_RFID.Inputs.Command", 1)
      on SwitchOn: SetTag("DB1_DatabaseAgv_RFID.Inputs.Command", 2)
      ProcessValue <- "DB1_DatabaseAgv_RFID.Inputs.Command"
   Button "Button_1" at 218,168 size 82x32; TextOff 'CONFIRMA GRAVAÇÃO'
      on Release: ResetBit("DB1_DatabaseAgv_RFID.Inputs.Start")
      on Press: SetBit("DB1_DatabaseAgv_RFID.Inputs.Start")
   TextField "Text field_1" at 17,146 size 99x13; Text 'ESCRITA/LEITURA'
   IOField "I/O field_4" at 22,52 size 35x20; FormatPattern 99
      ProcessValue <- "DB1_DatabaseAgv_RFID.Posto"
   IOField "I/O field_5" at 124,52 size 35x20; FormatPattern 99
      ProcessValue <- "DB1_DatabaseAgv_RFID.Comando"
   TextField "Text field_2" at 60,54 size 52x13; Text 'ESTAÇÃO'
   TextField "Text field_3" at 165,54 size 56x13; Text 'COMANDO'
   IOField "I/O field_6" at 231,52 size 35x20; FormatPattern 99
      ProcessValue <- "DB1_DatabaseAgv_RFID.Velocidade"
   TextField "Text field_4" at 271,55 size 51x13; Text 'VELOCID.'
   IOField "I/O field_7" at 23,113 size 35x20; FormatPattern 999
      ProcessValue <- "DB500_SinaisIhm_PostoRfid"
   TextField "Text field_5" at 70,7 size 190x18; Text 'CONFIGURAÇÃO DE TAGS RFID'
   TextField "Text field_6" at 111,34 size 89x15; Text 'VALORES LIDOS'
   TextField "Text field_7" at 84,94 size 151x15; Text 'VALORES PARA GRAVAÇÃO'
   IOField "I/O field_1" at 228,143 size 35x20; FormatPattern 999
      ProcessValue <- "DB500_SinaisIhm_ProcessoRfid"
   TextField "Text field_8" at 266,146 size 36x13; Text 'LINHA'
   IOField "I/O field_8" at 231,76 size 35x20; FormatPattern 99
      ProcessValue <- "DB1_DatabaseAgv_RFID.Processo"
   TextField "Text field_11" at 269,79 size 36x13; Text 'LINHA'
   Button "Button_2" at 120,167 size 71x32; TextOff 'RESET FALHA'
      on Release: ResetBit("DB500_SinaisIhm_ResetFalha_Rfid")
      on Press: SetBit("DB500_SinaisIhm_ResetFalha_Rfid")

Template "Template_2" 320x240
   Softkey "Softkey_F1" at 0,0 size 0x0; SoftkeyImage "Home"
      on KeyDown: ActivateScreen("00_Home", 0)
   Softkey "Softkey_F2" at 0,0 size 0x0; SoftkeyImage "Left_Arrow"
      on KeyDown: ActivateScreen("03_Manutecao", 0)

screen "10_InOutStatus" 320x240, template "Template_2"
   Circle "Circle_1" at 13,62 size 17x17
      Appearance <- "DB600_AgvSinais_Inputs.8DI_24V.I0.0"
   TextField "Text field_1" at 34,64 size 24x13; Text 'I0.0'
   Circle "Circle_2" at 90,62 size 17x17
      Appearance <- "DB600_AgvSinais_Inputs.8DI_24V.I0.1"
   TextField "Text field_2" at 111,64 size 24x13; Text 'I0.1'
   Circle "Circle_3" at 12,93 size 17x17
      Appearance <- "DB600_AgvSinais_Inputs.8DI_24V.I0.2"
   TextField "Text field_3" at 33,95 size 24x13; Text 'I0.2'
   Circle "Circle_4" at 90,94 size 17x17
      Appearance <- "DB600_AgvSinais_Inputs.8DI_24V.I0.3"
   TextField "Text field_4" at 111,96 size 24x13; Text 'I0.3'
   Circle "Circle_5" at 12,126 size 17x17
      Appearance <- "DB600_AgvSinais_Inputs.8DI_24V.I0.4"
   TextField "Text field_5" at 33,128 size 24x13; Text 'I0.4'
   Circle "Circle_6" at 90,128 size 17x17
      Appearance <- "DB600_AgvSinais_Inputs.8DI_24V.I0.5"
   TextField "Text field_6" at 111,130 size 24x13; Text 'I0.5'
   Circle "Circle_7" at 12,158 size 17x17
      Appearance <- "DB600_AgvSinais_Inputs.8DI_24V.I0.6"
   TextField "Text field_7" at 33,160 size 24x13; Text 'I0.6'
   Circle "Circle_8" at 89,159 size 17x17
      Appearance <- "DB600_AgvSinais_Inputs.8DI_24V.I0.7"
   TextField "Text field_8" at 110,161 size 24x13; Text 'I0.7'
   TextField "Text field_9" at 63,1 size 192x18; Text 'ENTRADA/SAIDAS DE SINAIS'
   TextField "Text field_10" at 24,32 size 98x20; Text '8DI x 24VDC'
   Circle "Circle_9" at 181,66 size 17x17
      Appearance <- "DB600_AgvSinais_Outputs.8DO_24V.Q0.0"
   TextField "Text field_11" at 202,68 size 27x13; Text 'Q0.0'
   Circle "Circle_10" at 258,67 size 17x17
      Appearance <- "DB600_AgvSinais_Outputs.8DO_24V.Q0.1"
   TextField "Text field_12" at 279,69 size 27x13; Text 'Q0.1'
   Circle "Circle_11" at 180,97 size 17x17
      Appearance <- "DB600_AgvSinais_Outputs.8DO_24V.Q0.2"
   TextField "Text field_13" at 201,99 size 27x13; Text 'Q0.2'
   Circle "Circle_12" at 258,99 size 17x17
      Appearance <- "DB600_AgvSinais_Outputs.8DO_24V.Q0.3"
   TextField "Text field_14" at 279,101 size 27x13; Text 'Q0.3'
   Circle "Circle_13" at 180,130 size 17x17
      Appearance <- "DB600_AgvSinais_Outputs.8DO_24V.Q0.4"
   TextField "Text field_15" at 201,132 size 27x13; Text 'Q0.4'
   Circle "Circle_14" at 258,133 size 17x17
      Appearance <- "DB600_AgvSinais_Outputs.8DO_24V.Q0.5"
   TextField "Text field_16" at 279,135 size 27x13; Text 'Q0.5'
   Circle "Circle_15" at 180,162 size 17x17
      Appearance <- "DB600_AgvSinais_Outputs.8DO_24V.Q0.6"
   TextField "Text field_17" at 201,164 size 27x13; Text 'Q0.6'
   Circle "Circle_16" at 257,164 size 17x17
      Appearance <- "DB600_AgvSinais_Outputs.8DO_24V.Q0.7"
   TextField "Text field_18" at 278,165 size 27x13; Text 'Q0.7'
   TextField "Text field_19" at 192,36 size 103x20; Text '8DO x 24VDC'
   IOField "I/O field_1" at 153,215 size 51x18; FormatPattern 99999
      ProcessValue <- "DB600_AgvSinais_Outputs.2AO x U ST.QW750"
   IOField "I/O field_2" at 261,215 size 51x18; FormatPattern 99999
      ProcessValue <- "DB600_AgvSinais_Outputs.2AO x U ST.QW752"
   TextField "Text field_20" at 114,214 size 35x16; Text 'Q750'
   TextField "Text field_21" at 224,214 size 35x16; Text 'Q752'
   TextField "Text field_22" at 187,202 size 60x13; Text '2AO x U ST'

screen "11_InStatusMotorDePasso" 320x240, template "Template_2"
   TextField "Text field_5" at 41,5 size 243x18; Text 'TELA DE STATUS DO MOTOR DE PASSO'
   GraphicView "Graphic view_1" at 7,45 size 95x85; Picture "Graphic_13"
   Circle "Circle_1" at 194,46 size 16x16
      Appearance <- "DB600_AgvSinais_Stepping_Motor.Inputs.Enabla_Drive"
   TextField "Text field_2" at 214,47 size 77x13; Text 'ENABLE DRIVE'
   Circle "Circle_2" at 194,66 size 16x16
      Appearance <- "DB600_AgvSinais_Stepping_Motor.Inputs.Stop"
   TextField "Text field_3" at 214,67 size 30x13; Text 'STOP'
   Circle "Circle_3" at 194,86 size 16x16
      Appearance <- "DB600_AgvSinais_Stepping_Motor.Inputs.Start Task"
   TextField "Text field_4" at 214,87 size 68x13; Text 'START TASK'
   TextField "Text field_6" at 195,108 size 26x13; Text 'OPM'
   Button "Button_1" at 223,152 size 76x32; TextOff 'PAGINA ANTERIOR'
      on Release: ActivateScreen("06_Status_Saida_MotorDePasso", 0)
   Button "Button_2" at 136,152 size 76x32; TextOff 'REALIZAR HOMING'
      on Release: ResetBit("DB1_DatabaseAgv_MotorDePasso.Inputs.StartHoming")
      on Press: SetBit("DB1_DatabaseAgv_MotorDePasso.Inputs.StartHoming")
   Button "Button_3" at 47,152 size 76x32; TextOff 'RESETAR FALHA'
      on Release: ResetBit("DB1_DatabaseAgv_MotorDePasso.Inputs.ResetFault")
      on Press: SetBit("DB1_DatabaseAgv_MotorDePasso.Inputs.ResetFault")
   IOField "I/O field_1" at 226,105 size 56x23; FormatPattern 999
      ProcessValue <- "DB600_AgvSinais_Stepping_Motor.Inputs.Opm"
   IOField "I/O field_5" at 109,203 size 210x35; FormatPattern ????????????????????????????????????????????
      ProcessValue <- "DB600_AgvSinais_Stepping_Motor.Mensagem"
   TextField "Text field_11" at 122,34 size 55x24; Text 'ACTUAL POSITION'
   IOField "I/O field_2" at 109,62 size 73x30; FormatPattern s9999999999
      ProcessValue <- "DB600_AgvSinais_Stepping_Motor.Outputs.ActualPosition"

screen "12_Alarms" 320x240, template "Template_2"
   AlarmView "Alarm view_1" at 3,5 size 309x191
   Button "Button_1" at 112,201 size 82x33; TextOff 'LIMPAR BUFFER'
      on Release: function_e14cd482(0)

screen "13_Diagnose" 320x240, template "Template_2"
   SysDiagControl "System diagnostics view_1" at 4,5 size 313x192
   Button "Button_1" at 114,203 size 82x33; TextOff 'LIMPAR BUFFER'
      on Release: function_e14cd482(0)

screen "14_StatusTakt" 320x240, template "Template_2"
   IOField "I/O field_5" at 0,164 size 319x35; FormatPattern ????????????????????????????????????????????
   TextField "Text field_1" at 45,39 size 62x15; Text 'BLOCO GET'
   Circle "Circle_6" at 36,68 size 18x18
      Appearance <- "DB703_ControleTakt_Out_Get_Error"
   TextField "Text field_13" at 63,67 size 45x18; Text 'ERROR'
   TextField "Text field_4" at 36,99 size 87x18; Text 'STATUS CODE'
   IOField "I/O field_1" at 42,123 size 62x23; FormatPattern FFFF
      ProcessValue <- "DB703_ControleTakt_Out_Get_Status"
   TextField "Text field_2" at 209,40 size 62x15; Text 'BLOCO GET'
   Circle "Circle_1" at 200,69 size 18x18
      Appearance <- "DB703_ControleTakt_Out_Set_Erro"
   TextField "Text field_3" at 227,68 size 45x18; Text 'ERROR'
   TextField "Text field_5" at 200,100 size 87x18; Text 'STATUS CODE'
   IOField "I/O field_2" at 206,124 size 62x23; FormatPattern FFFF
      ProcessValue <- "DB703_ControleTakt_Out_Set_Status"
   TextField "Text field_6" at 27,3 size 281x18; Text 'TELA DE STATUS DE COMUNICAÇÃO DO TAKT'
*)